FUNCTION derivcvar_M_p_t: LREAL
{ S7_Optimized_Access := 'true' }
    VAR_INPUT
        state: STATE;
    END_VAR

BEGIN
    derivcvar_M_p_t := 1.0;
END_FUNCTION
